# EPICS substitutions: iocBoot/iocvirPV/DPU07.substitutions
file "../../db/virAi.template"{ pattern
{DPU,	  num}
{07,	  0 }
{07,	  1 }
{07,	  2 }
{07,	  3 }
{07,	  4 }
{07,	  5 }
{07,	  6 }
{07,	  7 }
{07,	  8 }
{07,	  9 }
{07,	  10}
{07,	  11}
{07,	  12}
{07,	  13}
{07,	  14}
{07,	  15}
{07,	  16}
{07,	  17}
{07,	  18}
{07,	  19}
{07,	  20}
{07,	  21}
{07,	  22}
{07,	  23}
{07,	  24}
{07, 	  25}
{07,	  26}
{07,	  27}
{07,	  28}
{07,	  29}
{07,	  30}
{07,	  31}
{07,	  32}
{07,	  33}
{07,	  34}
{07,	  35}
{07,	  36}
{07,	  37}
{07,	  38}
{07,	  39}
{07,	  40}
{07,	  41}
{07,	  42}
{07,	  43}
{07,	  44}
{07,	  45}
{07,	  46}
{07,	  47}
{07,	  48}
{07,	  49}
{07,	  50}
{07,	  51}
{07,	  52}
{07,	  53}
{07,	  54}
{07,	  55}
{07,	  56}
{07,	  57}
{07,	  58}
{07,	  59}
{07,	  60}
{07,	  61}
{07,	  62}
{07, 	  63}
{07,      64}
{07,      65}
{07,      66}
{07,      67}
{07,      68}
{07,      69}
{07,      70}
{07,      71}
{07,      72}
{07,      73}
{07,      74}
{07,      75}
{07,      76}
{07,      77}
{07,      78}
{07,      79}
{07,      80}
{07,      81}
{07,      82}
{07,      83}
{07,      84}
{07,      85}
{07,      86}
{07,      87}
{07,      88}
{07,      89}
{07,      90}
{07,      91}
{07,      92}
{07,      93}
{07,      94}
{07,      95}
{07,      96}
{07,      97}
{07,      98}
{07,      99}
{07,     100}
{07,     101}
{07,     102}
{07,     103}
{07,     104}
{07,     105}
{07,     106}
{07,     107}
{07,     108}
{07,     109}
{07,     110}
{07,     111}
{07,     112}
{07,     113}
{07,     114}
{07,     115}
{07,     116}
{07,     117}
{07,     118}
{07,     119}
{07,     120}
{07,     121}
{07,     122}
{07,     123}
{07,     124}
{07,     125}
{07,     126}
{07,     127}
{07,     128}
{07,     129}
{07,     130}
{07,     131}
{07,     132}
{07,     133}
{07,     134}
{07,     135}
{07,     136}
{07,     137}
{07,     138}
{07,     139}
{07,     140}
{07,     141}
{07,     142}
{07,     143}
{07,     144}
{07,     145}
{07,     146}
{07,     147}
{07,     148}
{07,     149}
{07,     150}
{07,     151}
{07,     152}
{07,     153}
{07,     154}
{07,     155}
{07,     156}
{07,     157}
{07,     158}
{07,     159}
{07,     160}
{07,     161}
{07,     162}
{07,     163}
{07,     164}
{07,     165}
{07,     166}
{07,     167}
{07,     168}
{07,     169}
{07,     170}
{07,     171}
{07,     172}
{07,     173}
{07,     174}
{07,     175}
{07,     176}
{07,     177}
{07,     178}
{07,     179}
{07,     180}
{07,     181}
{07,     182}
{07,     183}
{07,     184}
{07,     185}
{07,     186}
{07,     187}
{07,     188}
{07,     189}
{07,     190}
{07,     191}
{07,     192}
{07,     193}
{07,     194}
{07,     195}
{07,     196}
{07,     197}
{07,     198}
{07,     199}
}
